DATA_BLOCK "ID_PE_Transport"
{ S7_Optimized_Access := 'TRUE' }
VERSION : 0.1
NON_RETAIN
"FB_PE_Transport"

BEGIN

END_DATA_BLOCK

